ABB RobotStudio station: team project (3) (1).rsstn

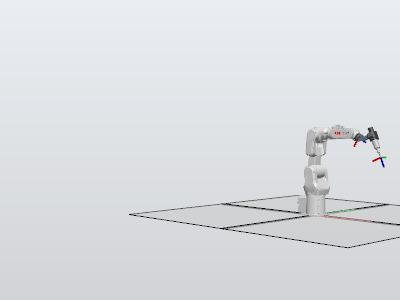
Station Station (saved by RobotStudio 24.1.10713.1)
Controller Controller6
  mechanical unit ROB_1: IRB1090_3_58__02, 6 joints, base frame (0, 0, 0) mm
Layout (positions relative to the parent item):
  - IRB1090_3_58__02 [mechanism, from %ABB.RobotStudio.Models.IRB1090%\IRB1090_3_58__01.rslib] at (0, 0, 0) mm; joint values [0.0119, 0.0672, -0.0877, -0.0466, 0.5055, 0.0083] (rad or m)
  - MyTool [mechanism, from Training Objects\myTool.rslib] at (375.14, 3.02, 592.7) mm, rotated rx -175.18 ry 62.14 rz -175.34 deg
Attachment: MyTool is attached to IRB1090_3_58__02 / Link6
Targets, tools, work objects and paths stored in the station, written as RAPID:
! task T_ROB1
MODULE CalibData
  PERS tooldata MyTool:=[TRUE,[[31.792631019,0,229.638935148],[0.945518576,0,0.325568154,0]],[1,[0,0,1],[1,0,0,0],0,0,0]];
ENDMODULE

